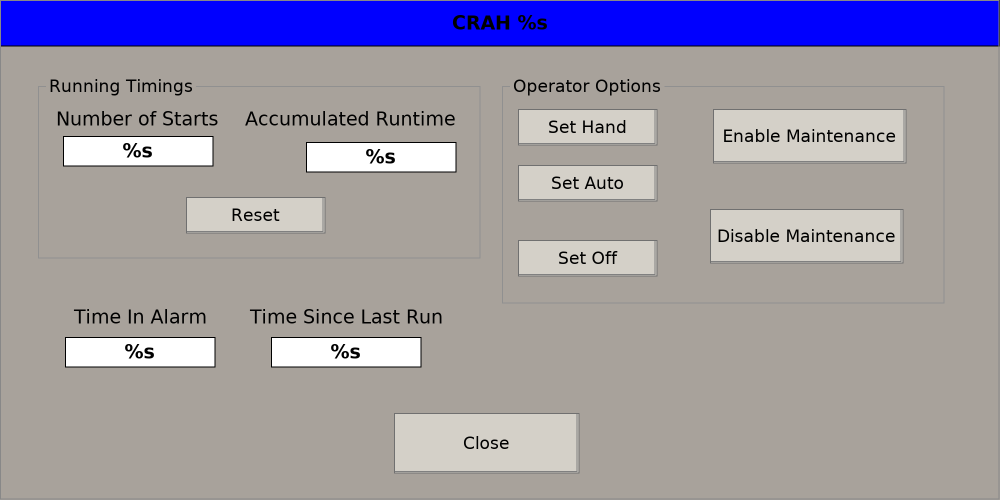
VISUALIZATION Dialog_CRAH  // 1000x500
VAR_IN_OUT
	sHeader : WSTRING;
	bCommonAlarm : BOOL;
	bIsolator1Alm :BOOL;
	bIsolator2Alm :BOOL;
	nSetControl :WORD;
	iNumStarts : WORD;
	sAccTime : STRING;
	sAlarmTime : STRING;
	sLastRunTime : STRING;
	bSetMaintenance : BOOL;
	bResetTimings : BOOL;
	
END_VAR
    Rectangle (0,0 1000x46), "CRAH %s", text variable: sHeader
    GroupBox (38,78 442x180), "Running Timings"
        Label (12,26 175x30), "Number of Starts"
        Rectangle (25,58 150x30), "%s", text variable: iNumStarts
        Label (202,26 221x30), "Accumulated Runtime"
        Rectangle (268,64 150x30), "%s", text variable: sAccTime
        Button (148,119 139x36), "Reset"
            OnMouseClick: execute { bResetTimings:=1; }
    GroupBox (502,78 442x225), "Operator Options"
        Label (12,26 175x30)
        Label (202,26 221x30)
        Button (16,31 139x36), "Set Hand"
            OnMouseClick: execute { nSetControl:=0; }
            OnMouseClick: CloseDialog Dialog=Dialog_CRAH, Result=OK, NumpadKeypadSet=True
        Button (16,87 139x36), "Set Auto"
            OnMouseClick: execute { bSetControl:=2; }
            OnMouseClick: CloseDialog Dialog=Dialog_CRAH, Result=OK, NumpadKeypadSet=True
        Button (16,162 139x36), "Set Off"
            OnMouseClick: execute { bSetControl:=1; }
            OnMouseClick: CloseDialog Dialog=Dialog_CRAH, Result=OK, NumpadKeypadSet=True
        Button (211,31 193x54), "Enable Maintenance"
            OnMouseClick: execute { bSetMaintenance:=1; }
            OnMouseClick: CloseDialog Dialog=Dialog_CRAH, Result=OK, NumpadKeypadSet=True
        Button (208,131 193x54), "Disable Maintenance"
            OnMouseClick: execute { bSetMaintenance:=0; }
            OnMouseClick: CloseDialog Dialog=Dialog_CRAH, Result=OK, NumpadKeypadSet=True
    Group (30,302 221x65)
        Rectangle (35,35 150x30), "%s", text variable: sAlarmTime
        Label (0,0 221x30), "Time In Alarm"
    Label (236,302 221x30), "Time Since Last Run"
    Rectangle (271,337 150x30), "%s", text variable: sLastRunTime
    Button (394,413 185x60), "Close"
        OnMouseClick: CloseDialog Dialog=Dialog_CRAH, Result=OK, NumpadKeypadSet=True
END_VISUALIZATION

(* stored: Version 1.1.0.1, ProductVersion 3.1.4024.12
   Visu Dialog_CRAH: Id {e3c68bac-9c3d-4bd7-ae79-5a69ea342bbb} *)
